FUNCTION_BLOCK Vendingmachine
VAR_INPUT
END_VAR
VAR_OUTPUT
END_VAR
VAR
	fbVending1: FB_Vending;
END_VAR

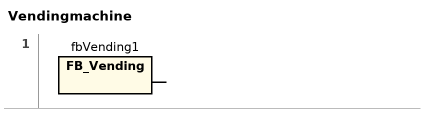
// NETWORK 1
fbVending1(); // FB_Vending

END_FUNCTION_BLOCK

(* stored: Version 1.1.0.1, ProductVersion 3.1.4022.16
   POU Vendingmachine: Id {a2f63a1d-53aa-4963-98fe-ae995ed7bc56}, SpecialFunc None *)
